// TIA Portal V15.1 export
// export: Created 2024-06-21T08:41:11.2554252Z, ExportSetting WithDefaults, DisplayName Totally Integrated Automation Portal, DisplayVersion V15.1 Update 5, DisplayName TIA Portal Openness, DisplayVersion V15.1 Update 5, DisplayName SINAMICS Startdrive Advanced, DisplayVersion V15.1, DisplayName G130, G150, S120, S150, SINAMICS MV, S210, DisplayVersion V15.1, DisplayName G110M, G120, G120C, G120D, G120P, DisplayVersion V15.1, DisplayName STEP 7 Professional, DisplayVersion V15.1 Update 5, DisplayName STEP 7 Safety, DisplayVersion V15.1, DisplayName WinCC Professional, DisplayVersion V15.1 Update 5, DisplayName SIMATIC Visualization Architect, DisplayVersion V15.1
FUNCTION "LGBHoist5Pos-MoviProPN-Config" : Void   // FC6695, FBD
TITLE = LMoveEPos-Config / LGBHoist5Pos-MoviProPN-Config
{ S7_Optimized_Access := 'FALSE' }
AUTHOR : VCC
FAMILY : Config
VERSION : 0.0.0.0
// =============================================================================
// Configuration MoveUnitEpos
// =============================================================================
// ============================================================================
// Configuration MoveUnitEpos
// ============================================================================
// stored: AutoNumber false, IsIECCheckEnabled false, SetENOAutomatically False, UDAEnableTagReadback false
   VAR_INPUT
      C_EnablePos1 : Bool;   // Pos 1 used
      C_EnablePos2 : Bool;   // Pos 2 used
      C_EnablePos3 : Bool;   // Pos 3 used
      C_EnablePos4 : Bool;   // Pos 4 used
      C_EnablePos5 : Bool;   // Pos 5 used / Pos 4 used
      C_EnablePosMaint : Bool;   // Pos Maintenance used / Pos 4 used
      C_BeltCheckSensor1Used : Bool;   // Belt check sensor 1 used
      C_BeltCheckSensor2Used : Bool;   // Belt check sensor 2 used
      C_2MotorsWithClutchDet : Bool;   // 2 motors with clutch detection
      C_OverTravelSetUsed : Bool;   // Overtravel set used
      C_OverTravelResUsed : Bool;   // Overtravel reset used
      C_MotorProtectionNc : Bool;   // Motor Protection NC contact
      C_MotorProtectionUsed : Bool;   // Motor Protection used
      C_MotionStopUsed : Bool;   // Motion Stop used
      C_EnableAlarmHW : Bool;   // Enable Alarm hardware (e.g. safetyswitch, motorprotector, detections)
      C_NotQuickStop : Bool;   // QuickStop function; When FALSE the QuickStop of the G120 is active
      C_ReleaseBrakeUsed : Bool;   // Release brake used
      C_ReferenceMotorCurrent : Real;   // Reference value for current, stored in P2002 ot the SINAMICS / Reference value for motor current
      C_ReferenceDriveCurrent : Real;   // Reference value for torque, stored in P2003 ot the SINAMICS / Reference value for drive current
      C_MaxRunTime : DInt;   // Time Delay-On Overtime Alarm (millisec)
      C_Acceleration : Int;   // EPOS MDI acceleration override / Acceleration in user units
      C_StopPos1 : DInt;   // Position Stop 1
      C_StopPos2 : DInt;   // Position Stop 2
      C_StopPos3 : DInt;   // Position Stop 3
      C_StopPos4 : DInt;   // Position Stop 4
      C_StopPos5 : DInt;   // Position Stop 4
      C_MaintenancePos : DInt;   // Maintenance Position
      C_TolerancePos : DInt;   // Tolerance Servo Position
      C_HWSubInput : HW_SUBMODULE;   // I/O
      C_HWSubOutput : HW_SUBMODULE;   // I/O
      C_HWSubController : HW_IO;   // Hardware identifier
   END_VAR
   VAR_IN_OUT
      IO_Config : "Hoist5Pos-MoviProPNConfig";   // Config
   END_VAR
BEGIN

REGION Network 1: **** 1 - Inputs **** Move Bit Config
   // Move Bit Config
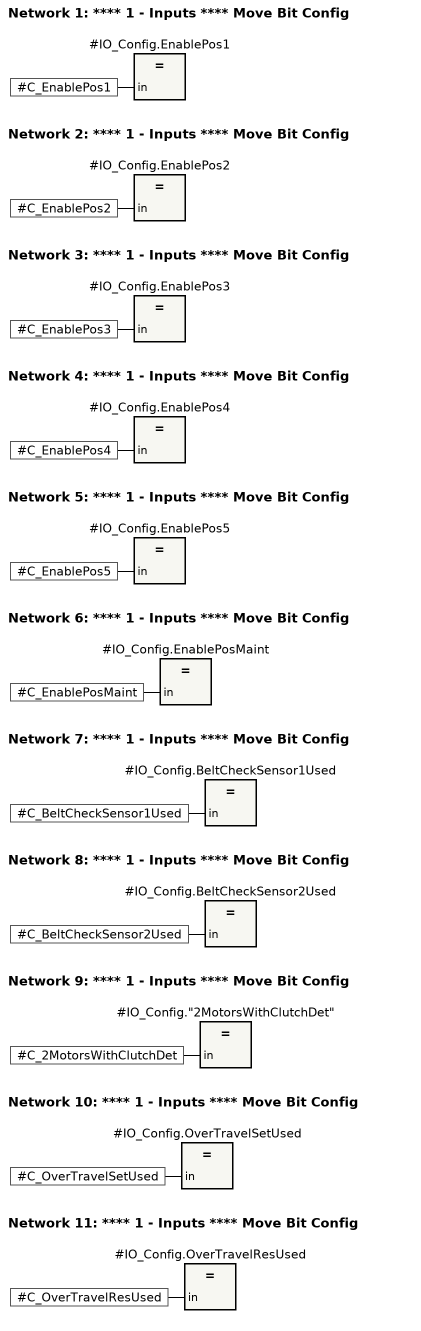
   #IO_Config.EnablePos1 := #C_EnablePos1;
END_REGION

REGION Network 2: **** 1 - Inputs **** Move Bit Config
   // Move Bit Config
   #IO_Config.EnablePos2 := #C_EnablePos2;
END_REGION

REGION Network 3: **** 1 - Inputs **** Move Bit Config
   // Move Bit Config
   #IO_Config.EnablePos3 := #C_EnablePos3;
END_REGION

REGION Network 4: **** 1 - Inputs **** Move Bit Config
   // Move Bit Config
   #IO_Config.EnablePos4 := #C_EnablePos4;
END_REGION

REGION Network 5: **** 1 - Inputs **** Move Bit Config
   // Move Bit Config
   #IO_Config.EnablePos5 := #C_EnablePos5;
END_REGION

REGION Network 6: **** 1 - Inputs **** Move Bit Config
   // Move Bit Config
   #IO_Config.EnablePosMaint := #C_EnablePosMaint;
END_REGION

REGION Network 7: **** 1 - Inputs **** Move Bit Config
   #IO_Config.BeltCheckSensor1Used := #C_BeltCheckSensor1Used;
END_REGION

REGION Network 8: **** 1 - Inputs **** Move Bit Config
   #IO_Config.BeltCheckSensor2Used := #C_BeltCheckSensor2Used;
END_REGION

REGION Network 9: **** 1 - Inputs **** Move Bit Config
   #IO_Config."2MotorsWithClutchDet" := #C_2MotorsWithClutchDet;
END_REGION

REGION Network 10: **** 1 - Inputs **** Move Bit Config
   #IO_Config.OverTravelSetUsed := #C_OverTravelSetUsed;
END_REGION

REGION Network 11: **** 1 - Inputs **** Move Bit Config
   #IO_Config.OverTravelResUsed := #C_OverTravelResUsed;
END_REGION

REGION Network 12: **** 1 - Inputs **** Move Bit Config
   // Move Bit Config
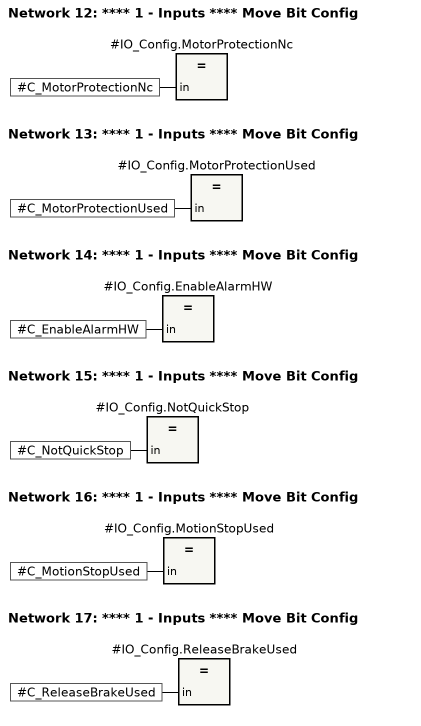
   #IO_Config.MotorProtectionNc := #C_MotorProtectionNc;
END_REGION

REGION Network 13: **** 1 - Inputs **** Move Bit Config
   // Move Bit Config
   #IO_Config.MotorProtectionUsed := #C_MotorProtectionUsed;
END_REGION

REGION Network 14: **** 1 - Inputs **** Move Bit Config
   // Move Bit Config
   #IO_Config.EnableAlarmHW := #C_EnableAlarmHW;
END_REGION

REGION Network 15: **** 1 - Inputs **** Move Bit Config
   // Move Bit Config
   #IO_Config.NotQuickStop := #C_NotQuickStop;
END_REGION

REGION Network 16: **** 1 - Inputs **** Move Bit Config
   // Move Bit Config
   #IO_Config.MotionStopUsed := #C_MotionStopUsed;
END_REGION

REGION Network 17: **** 1 - Inputs **** Move Bit Config
   // Move Bit Config
   #IO_Config.ReleaseBrakeUsed := #C_ReleaseBrakeUsed;
END_REGION

NETWORK
TITLE = **** 1 Inputs **** Move Config UDT
// Move Config
      L     #C_ReferenceMotorCurrent;
      T     #IO_Config.ReferenceMotorCurrent;
      L     #C_ReferenceDriveCurrent;
      T     #IO_Config.ReferenceDriveCurrent;
      L     #C_MaxRunTime;
      T     #IO_Config.MaxRunTime;
      L     #C_Acceleration;
      T     #IO_Config.Acceleration;
      L     #C_StopPos1;
      T     #IO_Config.StopPos1;
      L     #C_StopPos2;
      T     #IO_Config.StopPos2;
      L     #C_StopPos3;
      T     #IO_Config.StopPos3;
      L     #C_StopPos4;
      T     #IO_Config.StopPos4;
      L     #C_StopPos5;
      T     #IO_Config.StopPos5;
      L     #C_MaintenancePos;
      T     #IO_Config.MaintenancePos;
      L     #C_TolerancePos;
      T     #IO_Config.TolerancePos;
      L     #C_HWSubInput;
      T     #IO_Config.HWSubInput;
      L     #C_HWSubOutput;
      T     #IO_Config.HWSubOutput;
      L     #C_HWSubController;
      T     #IO_Config.HWSubController;
      NOP   0;
END_FUNCTION
